PROGRAM MAIN
VAR
	di1 AT %I* : BOOL;
	du1	AT %Q* : BOOL;
	ai1 AT %I* : INT;
	ao1 AT %Q* : INT;
	tmp1 AT %M* : REAL;
	counter : DINT; // 32 bit con segno
END_VAR

counter := counter + 1;

END_PROGRAM

(* stored: Version 1.1.0.1, ProductVersion 3.1.4024.12
   POU MAIN: Id {d3427bc8-5a67-46df-8492-351ac0137032}, SpecialFunc None *)
